FUNCTION_BLOCK T_UnsupportedEventHandler IMPLEMENTS I_UnsupportedEventHandler
VAR_INPUT
END_VAR
VAR_OUTPUT
END_VAR
VAR
END_VAR

END_FUNCTION_BLOCK

(* stored: Version 1.1.0.1, ProductVersion 3.1.4024.4
   POU T_UnsupportedEventHandler: Id {7946d37f-3e20-44e9-80d4-790f5f9013c7}, SpecialFunc None *)
